PROGRAM resetALL
VAR
END_VAR

IO.ElectroEntrar:=FALSE;
IO.ElectroPechar:=FALSE;
IO.ElectroPrensar:=FALSE;
IO.ElectroLiberar:=FALSE;
IO.ElectroAbrir:=FALSE;
IO.ElectroSair:=FALSE;

END_PROGRAM

(* stored: Version 1.1.0.1, ProductVersion 3.1.4024.9
   POU resetALL: Id {27617e08-9477-4ecd-8bc2-923926099a13}, SpecialFunc None *)
